FUNCTION TC_EventSeverityToString : STRING
VAR_INPUT
	eSeverity: TcEventSeverity;
END_VAR
VAR
	sSeverity:STRING;
END_VAR

CASE eSeverity OF
    TcEventSeverity.Verbose:
        sSeverity := 'Verbose';
    TcEventSeverity.Info:
        sSeverity := 'Info';
    TcEventSeverity.Warning:
        sSeverity := 'Warning';
    TcEventSeverity.Error:
        sSeverity := 'Error';
    TcEventSeverity.Critical:
        sSeverity := 'Critical';
ELSE
    sSeverity := 'Unknown';
END_CASE

TC_EventSeverityToString := sSeverity;

END_FUNCTION

(* stored: Version 1.1.0.1, ProductVersion 3.1.4024.15
   POU TC_EventSeverityToString: Id {08010551-e101-45c9-b921-e63e5661e3db}, SpecialFunc None *)
